{attribute 'strict'}
{attribute 'to_string'}
TYPE E_CylinderType :
(
    ThreePort_TwoPosition := 0,   // 3口2位
    FivePort_TwoPosition  := 1    // 5口2位
);
END_TYPE

(* stored: Version 1.1.0.1, ProductVersion 3.1.4024.15
   EnumerationTextList E_CylinderType: Id {d405793a-2849-4f2a-a742-95190b939d84} *)
